{attribute 'GeneratedUsingTerminal: EL3064-0000-0020'}
{attribute addProperty BoxType "EL3064-0000-0020"}
{attribute addProperty Id "StatusAT %I*Status_F2CE6D917ValueAT %I*INT2"}
{attribute addProperty CRC "1245267073"}
{attribute addProperty Size "9"}
TYPE AI_Standard_Channel_4A394481 :
STRUCT
	{attribute addProperty Name "Status"}
	Status AT %I* : Status_F2CE6D91;
	{attribute addProperty Name "Value"}
	Value AT %I* : INT;
END_STRUCT
END_TYPE

(* stored: Version 1.2.0.0, ProductVersion 3.1.4024.9
   DUT AI_Standard_Channel_4A394481: Id {ec4a9417-3f0c-405a-9564-498032dd1297} *)
